// TIA Portal V20 export
// export: Created 2025-12-01T14:57:47.0013054Z, ExportSetting None, DisplayName Totally Integrated Automation Portal, DisplayVersion V20 Update 3, DisplayName TIA Portal Openness, DisplayVersion V20 Update 3, DisplayName TIA Portal Version Control Interface, DisplayVersion V20 Update 3, DisplayName STEP 7 Professional, DisplayVersion V20 Update 3, DisplayName STEP 7 Safety, DisplayVersion V20 Update 2, DisplayName WinCC Basic/Comfort/Advanced, DisplayVersion V20 Update 3, DisplayName WinCC Professional, DisplayVersion V20 Update 3, DisplayName WinCC Unified, DisplayVersion V20 Update 3
DATA_BLOCK "DB921_DATOS_FECHA_HORA"   // DB921
{ S7_Optimized_Access := 'FALSE' }
AUTHOR : GENERAL
NAME : 20130301
VERSION : 3.0
// stored: AutoNumber false
   VAR
      SISTEMA : Date_And_Time;   // Variable provisional
      Actualizacion_1 : Date_And_Time;
      Incremento_Tiempo : Time;
      DI_Incremento_Tiempo : DInt;
      TIME_STAMP : String[20];
   END_VAR
BEGIN
END_DATA_BLOCK
